// TIA Portal project "Project3" (V16)

(* hardware
DEVICE "S7-1200 station_1"  S7-1200 Station
   slot 0: "Rack_0"  S7-1200 Rack  Rack  V1.0
   slot 1: "PLC_1"  CPU 1214C DC/DC/DC  6ES7 214-1AG40-0XB0  V4.4
*)

// ===== PLC "PLC_1"  CPU 1214C DC/DC/DC =====

VAR_GLOBAL   // PLC tag table "Default tag table"
   "START BUTTON" AT %I0.0 : Bool;
   "STOPBUTTON" AT %I0.1 : Bool;
   "RUN" AT %M0.2 : Bool;
   "MOTOR1" AT %Q0.3 : Bool;
   "MOTOR2" AT %Q0.4 : Bool;
   "DELAYED_STOP" AT %M0.5 : Bool;
   "TIMER_Q" AT %M0.6 : Bool;
   ""IEC_Timer_0_DB_1"" AT %M0.7 : Bool;
END_VAR

// folder: System blocks/Program resources

DATA_BLOCK "IEC_Timer_0_DB"   // DB1
{ S7_Optimized_Access := 'TRUE' }
AUTHOR : Simatic
FAMILY : IEC
NAME : IEC_TMR
VERSION : 1.0
// stored: InstanceOfName IEC_TIMER
"IEC_TIMER"
BEGIN
END_DATA_BLOCK

// folder: (top level)

ORGANIZATION_BLOCK "Main"   // OB1, LAD, ProgramCycle
TITLE = "Main Program Sweep (Cycle)"
{ S7_Optimized_Access := 'TRUE' }
VERSION : 0.1
   VAR_INPUT
      Initial_Call : Bool;   // Initial call of this OB
      Remanence : Bool;   // =True, if remanent data are available
   END_VAR
BEGIN

REGION Network 1
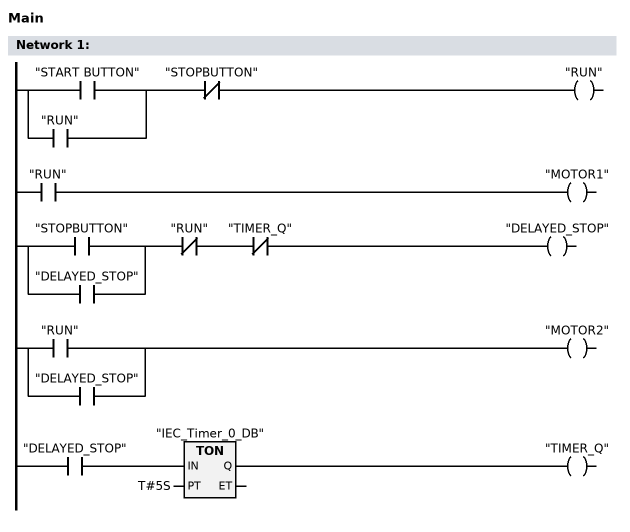
   "RUN" := ("START BUTTON" OR "RUN") AND NOT "STOPBUTTON";
   "MOTOR1" := "RUN";
   "DELAYED_STOP" := ("STOPBUTTON" OR "DELAYED_STOP") AND NOT "RUN" AND NOT "TIMER_Q";
   "MOTOR2" := "RUN" OR "DELAYED_STOP";
   "IEC_Timer_0_DB".TON(IN := "DELAYED_STOP", PT := T#5S);
   "TIMER_Q" := "IEC_Timer_0_DB".Q;
END_REGION
END_ORGANIZATION_BLOCK